TYPE structEstopDiag :
UNION
	iwordvalue:UINT;
	bitvalue:structSafetyEstopDiagBOOList;
END_UNION
END_TYPE

(* stored: Version 1.1.0.1, ProductVersion 3.1.4024.12
   DUT structEstopDiag: Id {c8d3e5c5-d85d-49d9-ac0b-8b27fdd8808e} *)
